//{attribute 'qualified_only'}
VAR_GLOBAL
	// PTM-03 on CH2, PTM-04 on CH1
	K2S17_E5_CH2_SerialRXBuffer : ComBuffer;
	K2S17_E5_CH2_SerialTXBuffer : ComBuffer;
	
	// Serial Terminal
	K2S17_E5_CH2_fbSerialLineControl: SerialLineControl;

	//SERIAL IO K2S17_E5_CH2 (EL6022)
	{attribute	'TcLinkTo'	:=	'.Status:=TIID^Device 1 (EtherCAT)^Term 1 (EK1200)^Term 2 (EK1122)^Hoffman Box Vac EK1 (EK1100)^E5 (EL6022)^COM Inputs Channel 2^Status;
								 .D[0]:=TIID^Device 1 (EtherCAT)^Term 1 (EK1200)^Term 2 (EK1122)^Hoffman Box Vac EK1 (EK1100)^E5 (EL6022)^COM Inputs Channel 2^Data In 0;
								 .D[1]:=TIID^Device 1 (EtherCAT)^Term 1 (EK1200)^Term 2 (EK1122)^Hoffman Box Vac EK1 (EK1100)^E5 (EL6022)^COM Inputs Channel 2^Data In 1;
								 .D[2]:=TIID^Device 1 (EtherCAT)^Term 1 (EK1200)^Term 2 (EK1122)^Hoffman Box Vac EK1 (EK1100)^E5 (EL6022)^COM Inputs Channel 2^Data In 2;
								 .D[3]:=TIID^Device 1 (EtherCAT)^Term 1 (EK1200)^Term 2 (EK1122)^Hoffman Box Vac EK1 (EK1100)^E5 (EL6022)^COM Inputs Channel 2^Data In 3;
								 .D[4]:=TIID^Device 1 (EtherCAT)^Term 1 (EK1200)^Term 2 (EK1122)^Hoffman Box Vac EK1 (EK1100)^E5 (EL6022)^COM Inputs Channel 2^Data In 4;
								 .D[5]:=TIID^Device 1 (EtherCAT)^Term 1 (EK1200)^Term 2 (EK1122)^Hoffman Box Vac EK1 (EK1100)^E5 (EL6022)^COM Inputs Channel 2^Data In 5;
								 .D[6]:=TIID^Device 1 (EtherCAT)^Term 1 (EK1200)^Term 2 (EK1122)^Hoffman Box Vac EK1 (EK1100)^E5 (EL6022)^COM Inputs Channel 2^Data In 6;
								 .D[7]:=TIID^Device 1 (EtherCAT)^Term 1 (EK1200)^Term 2 (EK1122)^Hoffman Box Vac EK1 (EK1100)^E5 (EL6022)^COM Inputs Channel 2^Data In 7;
								 .D[8]:=TIID^Device 1 (EtherCAT)^Term 1 (EK1200)^Term 2 (EK1122)^Hoffman Box Vac EK1 (EK1100)^E5 (EL6022)^COM Inputs Channel 2^Data In 8;
								 .D[9]:=TIID^Device 1 (EtherCAT)^Term 1 (EK1200)^Term 2 (EK1122)^Hoffman Box Vac EK1 (EK1100)^E5 (EL6022)^COM Inputs Channel 2^Data In 9;
								 .D[10]:=TIID^Device 1 (EtherCAT)^Term 1 (EK1200)^Term 2 (EK1122)^Hoffman Box Vac EK1 (EK1100)^E5 (EL6022)^COM Inputs Channel 2^Data In 10;
								 .D[11]:=TIID^Device 1 (EtherCAT)^Term 1 (EK1200)^Term 2 (EK1122)^Hoffman Box Vac EK1 (EK1100)^E5 (EL6022)^COM Inputs Channel 2^Data In 11;
								 .D[12]:=TIID^Device 1 (EtherCAT)^Term 1 (EK1200)^Term 2 (EK1122)^Hoffman Box Vac EK1 (EK1100)^E5 (EL6022)^COM Inputs Channel 2^Data In 12;
								 .D[13]:=TIID^Device 1 (EtherCAT)^Term 1 (EK1200)^Term 2 (EK1122)^Hoffman Box Vac EK1 (EK1100)^E5 (EL6022)^COM Inputs Channel 2^Data In 13;
								 .D[14]:=TIID^Device 1 (EtherCAT)^Term 1 (EK1200)^Term 2 (EK1122)^Hoffman Box Vac EK1 (EK1100)^E5 (EL6022)^COM Inputs Channel 2^Data In 14;
								 .D[15]:=TIID^Device 1 (EtherCAT)^Term 1 (EK1200)^Term 2 (EK1122)^Hoffman Box Vac EK1 (EK1100)^E5 (EL6022)^COM Inputs Channel 2^Data In 15;
								 .D[16]:=TIID^Device 1 (EtherCAT)^Term 1 (EK1200)^Term 2 (EK1122)^Hoffman Box Vac EK1 (EK1100)^E5 (EL6022)^COM Inputs Channel 2^Data In 16;
								 .D[17]:=TIID^Device 1 (EtherCAT)^Term 1 (EK1200)^Term 2 (EK1122)^Hoffman Box Vac EK1 (EK1100)^E5 (EL6022)^COM Inputs Channel 2^Data In 17;
								 .D[18]:=TIID^Device 1 (EtherCAT)^Term 1 (EK1200)^Term 2 (EK1122)^Hoffman Box Vac EK1 (EK1100)^E5 (EL6022)^COM Inputs Channel 2^Data In 18;
								 .D[19]:=TIID^Device 1 (EtherCAT)^Term 1 (EK1200)^Term 2 (EK1122)^Hoffman Box Vac EK1 (EK1100)^E5 (EL6022)^COM Inputs Channel 2^Data In 19;
								 .D[20]:=TIID^Device 1 (EtherCAT)^Term 1 (EK1200)^Term 2 (EK1122)^Hoffman Box Vac EK1 (EK1100)^E5 (EL6022)^COM Inputs Channel 2^Data In 20;
								 .D[21]:=TIID^Device 1 (EtherCAT)^Term 1 (EK1200)^Term 2 (EK1122)^Hoffman Box Vac EK1 (EK1100)^E5 (EL6022)^COM Inputs Channel 2^Data In 21
	'}
	K2S17_E5_CH2_stComIn		AT %I*	:	EL6inData22B; 
	{attribute	'TcLinkTo'	:=	'.Ctrl:=TIID^Device 1 (EtherCAT)^Term 1 (EK1200)^Term 2 (EK1122)^Hoffman Box Vac EK1 (EK1100)^E5 (EL6022)^COM Outputs Channel 2^Ctrl;
								 .D[0]:=TIID^Device 1 (EtherCAT)^Term 1 (EK1200)^Term 2 (EK1122)^Hoffman Box Vac EK1 (EK1100)^E5 (EL6022)^COM Outputs Channel 2^Data Out 0;
								 .D[1]:=TIID^Device 1 (EtherCAT)^Term 1 (EK1200)^Term 2 (EK1122)^Hoffman Box Vac EK1 (EK1100)^E5 (EL6022)^COM Outputs Channel 2^Data Out 1;
								 .D[2]:=TIID^Device 1 (EtherCAT)^Term 1 (EK1200)^Term 2 (EK1122)^Hoffman Box Vac EK1 (EK1100)^E5 (EL6022)^COM Outputs Channel 2^Data Out 2;
								 .D[3]:=TIID^Device 1 (EtherCAT)^Term 1 (EK1200)^Term 2 (EK1122)^Hoffman Box Vac EK1 (EK1100)^E5 (EL6022)^COM Outputs Channel 2^Data Out 3;
								 .D[4]:=TIID^Device 1 (EtherCAT)^Term 1 (EK1200)^Term 2 (EK1122)^Hoffman Box Vac EK1 (EK1100)^E5 (EL6022)^COM Outputs Channel 2^Data Out 4;
								 .D[5]:=TIID^Device 1 (EtherCAT)^Term 1 (EK1200)^Term 2 (EK1122)^Hoffman Box Vac EK1 (EK1100)^E5 (EL6022)^COM Outputs Channel 2^Data Out 5;
								 .D[6]:=TIID^Device 1 (EtherCAT)^Term 1 (EK1200)^Term 2 (EK1122)^Hoffman Box Vac EK1 (EK1100)^E5 (EL6022)^COM Outputs Channel 2^Data Out 6;
								 .D[7]:=TIID^Device 1 (EtherCAT)^Term 1 (EK1200)^Term 2 (EK1122)^Hoffman Box Vac EK1 (EK1100)^E5 (EL6022)^COM Outputs Channel 2^Data Out 7;
								 .D[8]:=TIID^Device 1 (EtherCAT)^Term 1 (EK1200)^Term 2 (EK1122)^Hoffman Box Vac EK1 (EK1100)^E5 (EL6022)^COM Outputs Channel 2^Data Out 8;
								 .D[9]:=TIID^Device 1 (EtherCAT)^Term 1 (EK1200)^Term 2 (EK1122)^Hoffman Box Vac EK1 (EK1100)^E5 (EL6022)^COM Outputs Channel 2^Data Out 9;
								 .D[10]:=TIID^Device 1 (EtherCAT)^Term 1 (EK1200)^Term 2 (EK1122)^Hoffman Box Vac EK1 (EK1100)^E5 (EL6022)^COM Outputs Channel 2^Data Out 10;
								 .D[11]:=TIID^Device 1 (EtherCAT)^Term 1 (EK1200)^Term 2 (EK1122)^Hoffman Box Vac EK1 (EK1100)^E5 (EL6022)^COM Outputs Channel 2^Data Out 11;
								 .D[12]:=TIID^Device 1 (EtherCAT)^Term 1 (EK1200)^Term 2 (EK1122)^Hoffman Box Vac EK1 (EK1100)^E5 (EL6022)^COM Outputs Channel 2^Data Out 12;
								 .D[13]:=TIID^Device 1 (EtherCAT)^Term 1 (EK1200)^Term 2 (EK1122)^Hoffman Box Vac EK1 (EK1100)^E5 (EL6022)^COM Outputs Channel 2^Data Out 13;
								 .D[14]:=TIID^Device 1 (EtherCAT)^Term 1 (EK1200)^Term 2 (EK1122)^Hoffman Box Vac EK1 (EK1100)^E5 (EL6022)^COM Outputs Channel 2^Data Out 14;
								 .D[15]:=TIID^Device 1 (EtherCAT)^Term 1 (EK1200)^Term 2 (EK1122)^Hoffman Box Vac EK1 (EK1100)^E5 (EL6022)^COM Outputs Channel 2^Data Out 15;
								 .D[16]:=TIID^Device 1 (EtherCAT)^Term 1 (EK1200)^Term 2 (EK1122)^Hoffman Box Vac EK1 (EK1100)^E5 (EL6022)^COM Outputs Channel 2^Data Out 16;
								 .D[17]:=TIID^Device 1 (EtherCAT)^Term 1 (EK1200)^Term 2 (EK1122)^Hoffman Box Vac EK1 (EK1100)^E5 (EL6022)^COM Outputs Channel 2^Data Out 17;
								 .D[18]:=TIID^Device 1 (EtherCAT)^Term 1 (EK1200)^Term 2 (EK1122)^Hoffman Box Vac EK1 (EK1100)^E5 (EL6022)^COM Outputs Channel 2^Data Out 18;
								 .D[19]:=TIID^Device 1 (EtherCAT)^Term 1 (EK1200)^Term 2 (EK1122)^Hoffman Box Vac EK1 (EK1100)^E5 (EL6022)^COM Outputs Channel 2^Data Out 19;
								 .D[20]:=TIID^Device 1 (EtherCAT)^Term 1 (EK1200)^Term 2 (EK1122)^Hoffman Box Vac EK1 (EK1100)^E5 (EL6022)^COM Outputs Channel 2^Data Out 20;
								 .D[21]:=TIID^Device 1 (EtherCAT)^Term 1 (EK1200)^Term 2 (EK1122)^Hoffman Box Vac EK1 (EK1100)^E5 (EL6022)^COM Outputs Channel 2^Data Out 21
	'}
	K2S17_E5_CH2_stComOut		AT %Q*	:	EL6outData22B;
	
	
	
	// PTM-04 on CH1
	K2S17_E5_CH1_SerialRXBuffer : ComBuffer;
	K2S17_E5_CH1_SerialTXBuffer : ComBuffer;
	
	// Serial Terminal
	K2S17_E5_CH1_fbSerialLineControl: SerialLineControl;

	//SERIAL IO K2S17_E5_CH1 (EL6022)
	{attribute	'TcLinkTo'	:=	'.Status:=TIID^Device 1 (EtherCAT)^Term 1 (EK1200)^Term 2 (EK1122)^Hoffman Box Vac EK1 (EK1100)^E5 (EL6022)^COM Inputs Channel 1^Status;
								 .D[0]:=TIID^Device 1 (EtherCAT)^Term 1 (EK1200)^Term 2 (EK1122)^Hoffman Box Vac EK1 (EK1100)^E5 (EL6022)^COM Inputs Channel 1^Data In 0;
								 .D[1]:=TIID^Device 1 (EtherCAT)^Term 1 (EK1200)^Term 2 (EK1122)^Hoffman Box Vac EK1 (EK1100)^E5 (EL6022)^COM Inputs Channel 1^Data In 1;
								 .D[2]:=TIID^Device 1 (EtherCAT)^Term 1 (EK1200)^Term 2 (EK1122)^Hoffman Box Vac EK1 (EK1100)^E5 (EL6022)^COM Inputs Channel 1^Data In 2;
								 .D[3]:=TIID^Device 1 (EtherCAT)^Term 1 (EK1200)^Term 2 (EK1122)^Hoffman Box Vac EK1 (EK1100)^E5 (EL6022)^COM Inputs Channel 1^Data In 3;
								 .D[4]:=TIID^Device 1 (EtherCAT)^Term 1 (EK1200)^Term 2 (EK1122)^Hoffman Box Vac EK1 (EK1100)^E5 (EL6022)^COM Inputs Channel 1^Data In 4;
								 .D[5]:=TIID^Device 1 (EtherCAT)^Term 1 (EK1200)^Term 2 (EK1122)^Hoffman Box Vac EK1 (EK1100)^E5 (EL6022)^COM Inputs Channel 1^Data In 5;
								 .D[6]:=TIID^Device 1 (EtherCAT)^Term 1 (EK1200)^Term 2 (EK1122)^Hoffman Box Vac EK1 (EK1100)^E5 (EL6022)^COM Inputs Channel 1^Data In 6;
								 .D[7]:=TIID^Device 1 (EtherCAT)^Term 1 (EK1200)^Term 2 (EK1122)^Hoffman Box Vac EK1 (EK1100)^E5 (EL6022)^COM Inputs Channel 1^Data In 7;
								 .D[8]:=TIID^Device 1 (EtherCAT)^Term 1 (EK1200)^Term 2 (EK1122)^Hoffman Box Vac EK1 (EK1100)^E5 (EL6022)^COM Inputs Channel 1^Data In 8;
								 .D[9]:=TIID^Device 1 (EtherCAT)^Term 1 (EK1200)^Term 2 (EK1122)^Hoffman Box Vac EK1 (EK1100)^E5 (EL6022)^COM Inputs Channel 1^Data In 9;
								 .D[10]:=TIID^Device 1 (EtherCAT)^Term 1 (EK1200)^Term 2 (EK1122)^Hoffman Box Vac EK1 (EK1100)^E5 (EL6022)^COM Inputs Channel 1^Data In 10;
								 .D[11]:=TIID^Device 1 (EtherCAT)^Term 1 (EK1200)^Term 2 (EK1122)^Hoffman Box Vac EK1 (EK1100)^E5 (EL6022)^COM Inputs Channel 1^Data In 11;
								 .D[12]:=TIID^Device 1 (EtherCAT)^Term 1 (EK1200)^Term 2 (EK1122)^Hoffman Box Vac EK1 (EK1100)^E5 (EL6022)^COM Inputs Channel 1^Data In 12;
								 .D[13]:=TIID^Device 1 (EtherCAT)^Term 1 (EK1200)^Term 2 (EK1122)^Hoffman Box Vac EK1 (EK1100)^E5 (EL6022)^COM Inputs Channel 1^Data In 13;
								 .D[14]:=TIID^Device 1 (EtherCAT)^Term 1 (EK1200)^Term 2 (EK1122)^Hoffman Box Vac EK1 (EK1100)^E5 (EL6022)^COM Inputs Channel 1^Data In 14;
								 .D[15]:=TIID^Device 1 (EtherCAT)^Term 1 (EK1200)^Term 2 (EK1122)^Hoffman Box Vac EK1 (EK1100)^E5 (EL6022)^COM Inputs Channel 1^Data In 15;
								 .D[16]:=TIID^Device 1 (EtherCAT)^Term 1 (EK1200)^Term 2 (EK1122)^Hoffman Box Vac EK1 (EK1100)^E5 (EL6022)^COM Inputs Channel 1^Data In 16;
								 .D[17]:=TIID^Device 1 (EtherCAT)^Term 1 (EK1200)^Term 2 (EK1122)^Hoffman Box Vac EK1 (EK1100)^E5 (EL6022)^COM Inputs Channel 1^Data In 17;
								 .D[18]:=TIID^Device 1 (EtherCAT)^Term 1 (EK1200)^Term 2 (EK1122)^Hoffman Box Vac EK1 (EK1100)^E5 (EL6022)^COM Inputs Channel 1^Data In 18;
								 .D[19]:=TIID^Device 1 (EtherCAT)^Term 1 (EK1200)^Term 2 (EK1122)^Hoffman Box Vac EK1 (EK1100)^E5 (EL6022)^COM Inputs Channel 1^Data In 19;
								 .D[20]:=TIID^Device 1 (EtherCAT)^Term 1 (EK1200)^Term 2 (EK1122)^Hoffman Box Vac EK1 (EK1100)^E5 (EL6022)^COM Inputs Channel 1^Data In 20;
								 .D[21]:=TIID^Device 1 (EtherCAT)^Term 1 (EK1200)^Term 2 (EK1122)^Hoffman Box Vac EK1 (EK1100)^E5 (EL6022)^COM Inputs Channel 1^Data In 21
	'}
	K2S17_E5_CH1_stComIn		AT %I*	:	EL6inData22B; 
	{attribute	'TcLinkTo'	:=	'.Ctrl:=TIID^Device 1 (EtherCAT)^Term 1 (EK1200)^Term 2 (EK1122)^Hoffman Box Vac EK1 (EK1100)^E5 (EL6022)^COM Outputs Channel 1^Ctrl;
								 .D[0]:=TIID^Device 1 (EtherCAT)^Term 1 (EK1200)^Term 2 (EK1122)^Hoffman Box Vac EK1 (EK1100)^E5 (EL6022)^COM Outputs Channel 1^Data Out 0;
								 .D[1]:=TIID^Device 1 (EtherCAT)^Term 1 (EK1200)^Term 2 (EK1122)^Hoffman Box Vac EK1 (EK1100)^E5 (EL6022)^COM Outputs Channel 1^Data Out 1;
								 .D[2]:=TIID^Device 1 (EtherCAT)^Term 1 (EK1200)^Term 2 (EK1122)^Hoffman Box Vac EK1 (EK1100)^E5 (EL6022)^COM Outputs Channel 1^Data Out 2;
								 .D[3]:=TIID^Device 1 (EtherCAT)^Term 1 (EK1200)^Term 2 (EK1122)^Hoffman Box Vac EK1 (EK1100)^E5 (EL6022)^COM Outputs Channel 1^Data Out 3;
								 .D[4]:=TIID^Device 1 (EtherCAT)^Term 1 (EK1200)^Term 2 (EK1122)^Hoffman Box Vac EK1 (EK1100)^E5 (EL6022)^COM Outputs Channel 1^Data Out 4;
								 .D[5]:=TIID^Device 1 (EtherCAT)^Term 1 (EK1200)^Term 2 (EK1122)^Hoffman Box Vac EK1 (EK1100)^E5 (EL6022)^COM Outputs Channel 1^Data Out 5;
								 .D[6]:=TIID^Device 1 (EtherCAT)^Term 1 (EK1200)^Term 2 (EK1122)^Hoffman Box Vac EK1 (EK1100)^E5 (EL6022)^COM Outputs Channel 1^Data Out 6;
								 .D[7]:=TIID^Device 1 (EtherCAT)^Term 1 (EK1200)^Term 2 (EK1122)^Hoffman Box Vac EK1 (EK1100)^E5 (EL6022)^COM Outputs Channel 1^Data Out 7;
								 .D[8]:=TIID^Device 1 (EtherCAT)^Term 1 (EK1200)^Term 2 (EK1122)^Hoffman Box Vac EK1 (EK1100)^E5 (EL6022)^COM Outputs Channel 1^Data Out 8;
								 .D[9]:=TIID^Device 1 (EtherCAT)^Term 1 (EK1200)^Term 2 (EK1122)^Hoffman Box Vac EK1 (EK1100)^E5 (EL6022)^COM Outputs Channel 1^Data Out 9;
								 .D[10]:=TIID^Device 1 (EtherCAT)^Term 1 (EK1200)^Term 2 (EK1122)^Hoffman Box Vac EK1 (EK1100)^E5 (EL6022)^COM Outputs Channel 1^Data Out 10;
								 .D[11]:=TIID^Device 1 (EtherCAT)^Term 1 (EK1200)^Term 2 (EK1122)^Hoffman Box Vac EK1 (EK1100)^E5 (EL6022)^COM Outputs Channel 1^Data Out 11;
								 .D[12]:=TIID^Device 1 (EtherCAT)^Term 1 (EK1200)^Term 2 (EK1122)^Hoffman Box Vac EK1 (EK1100)^E5 (EL6022)^COM Outputs Channel 1^Data Out 12;
								 .D[13]:=TIID^Device 1 (EtherCAT)^Term 1 (EK1200)^Term 2 (EK1122)^Hoffman Box Vac EK1 (EK1100)^E5 (EL6022)^COM Outputs Channel 1^Data Out 13;
								 .D[14]:=TIID^Device 1 (EtherCAT)^Term 1 (EK1200)^Term 2 (EK1122)^Hoffman Box Vac EK1 (EK1100)^E5 (EL6022)^COM Outputs Channel 1^Data Out 14;
								 .D[15]:=TIID^Device 1 (EtherCAT)^Term 1 (EK1200)^Term 2 (EK1122)^Hoffman Box Vac EK1 (EK1100)^E5 (EL6022)^COM Outputs Channel 1^Data Out 15;
								 .D[16]:=TIID^Device 1 (EtherCAT)^Term 1 (EK1200)^Term 2 (EK1122)^Hoffman Box Vac EK1 (EK1100)^E5 (EL6022)^COM Outputs Channel 1^Data Out 16;
								 .D[17]:=TIID^Device 1 (EtherCAT)^Term 1 (EK1200)^Term 2 (EK1122)^Hoffman Box Vac EK1 (EK1100)^E5 (EL6022)^COM Outputs Channel 1^Data Out 17;
								 .D[18]:=TIID^Device 1 (EtherCAT)^Term 1 (EK1200)^Term 2 (EK1122)^Hoffman Box Vac EK1 (EK1100)^E5 (EL6022)^COM Outputs Channel 1^Data Out 18;
								 .D[19]:=TIID^Device 1 (EtherCAT)^Term 1 (EK1200)^Term 2 (EK1122)^Hoffman Box Vac EK1 (EK1100)^E5 (EL6022)^COM Outputs Channel 1^Data Out 19;
								 .D[20]:=TIID^Device 1 (EtherCAT)^Term 1 (EK1200)^Term 2 (EK1122)^Hoffman Box Vac EK1 (EK1100)^E5 (EL6022)^COM Outputs Channel 1^Data Out 20;
								 .D[21]:=TIID^Device 1 (EtherCAT)^Term 1 (EK1200)^Term 2 (EK1122)^Hoffman Box Vac EK1 (EK1100)^E5 (EL6022)^COM Outputs Channel 1^Data Out 21
	'}
	K2S17_E5_CH1_stComOut		AT %Q*	:	EL6outData22B;
END_VAR

(* stored: Version 1.1.0.1, ProductVersion 3.1.4022.18
   GVL GVL_COM: Id {d3571159-1af9-459a-a3b2-17c060e0c123} *)
